// TIA Portal V20 export
FUNCTION "ManOperationCm_typeTwoWayActuatorInterface" : Void   // FC65, LAD
// stored: SetENOAutomatically false
   VAR_INPUT
      disableUnit : Bool;
   END_VAR
   VAR_OUTPUT
      Status : Word;
      errorID : Word;
   END_VAR
   VAR_IN_OUT
      manualOperationEm : "LAF_typeManEm";
      manualOperationEmArea : "LAF_typeManOperationArea";
      manualOperationCms : "LAF_typeManOperation";
      twoWayAcutor : "LBC_typeTwoWayActuatorInterface";
   END_VAR
BEGIN

REGION Network 1: Manual Operation Cm - typeTwoWayActuatorInterface
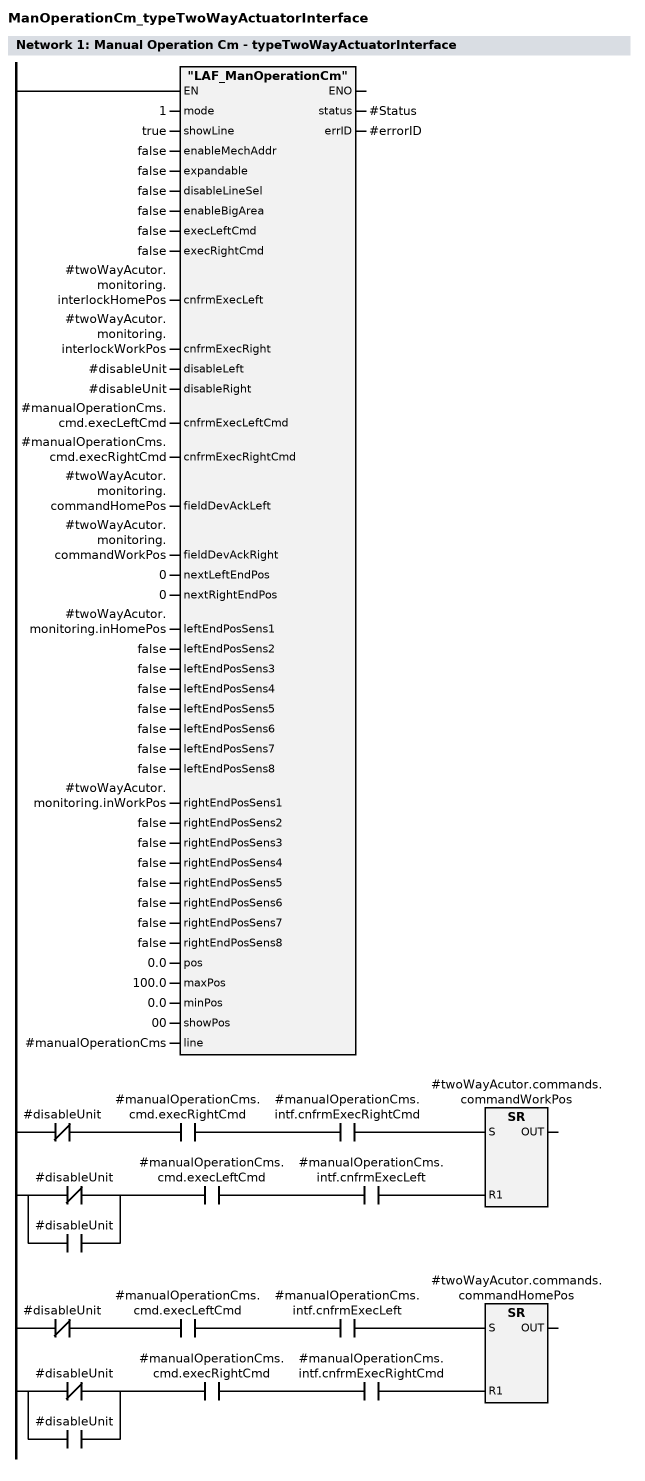
   RUNG wire#powerrail
      "LAF_ManOperationCm"(mode := 1, showLine := true, enableMechAddr := false, expandable := false, disableLineSel := false, enableBigArea := false, execLeftCmd := false, execRightCmd := false, cnfrmExecLeft := #twoWayAcutor.monitoring.interlockHomePos, cnfrmExecRight := #twoWayAcutor.monitoring.interlockWorkPos, disableLeft := #disableUnit, disableRight := #disableUnit, cnfrmExecLeftCmd := #manualOperationCms.cmd.execLeftCmd, cnfrmExecRightCmd := #manualOperationCms.cmd.execRightCmd, fieldDevAckLeft := #twoWayAcutor.monitoring.commandHomePos, fieldDevAckRight := #twoWayAcutor.monitoring.commandWorkPos, nextLeftEndPos := 0, nextRightEndPos := 0, leftEndPosSens1 := #twoWayAcutor.monitoring.inHomePos, leftEndPosSens2 := false, leftEndPosSens3 := false, leftEndPosSens4 := false, leftEndPosSens5 := false, leftEndPosSens6 := false, leftEndPosSens7 := false, leftEndPosSens8 := false, rightEndPosSens1 := #twoWayAcutor.monitoring.inWorkPos, rightEndPosSens2 := false, rightEndPosSens3 := false, rightEndPosSens4 := false, rightEndPosSens5 := false, rightEndPosSens6 := false, rightEndPosSens7 := false, rightEndPosSens8 := false, pos := 0.0, maxPos := 100.0, minPos := 0.0, showPos := 00, line := #manualOperationCms, status => #Status, errID => #errorID)
   END_RUNG
   RUNG wire#powerrail
      I_Contact( #disableUnit )
      Contact( #manualOperationCms.cmd.execRightCmd )
      Contact( #manualOperationCms.intf.cnfrmExecRightCmd )
      S_SR(operand := #twoWayAcutor.commands.commandWorkPos, r1 := wire#w2)
   END_RUNG
   RUNG wire#powerrail
      I_Contact( #disableUnit )
      wire#w1
      Contact( #manualOperationCms.cmd.execLeftCmd )
      Contact( #manualOperationCms.intf.cnfrmExecLeft )
   END_RUNG wire#w2
   RUNG wire#powerrail
      Contact( #disableUnit )
   END_RUNG wire#w1
   RUNG wire#powerrail
      I_Contact( #disableUnit )
      Contact( #manualOperationCms.cmd.execLeftCmd )
      Contact( #manualOperationCms.intf.cnfrmExecLeft )
      S_SR(operand := #twoWayAcutor.commands.commandHomePos, r1 := wire#w4)
   END_RUNG
   RUNG wire#powerrail
      I_Contact( #disableUnit )
      wire#w3
      Contact( #manualOperationCms.cmd.execRightCmd )
      Contact( #manualOperationCms.intf.cnfrmExecRightCmd )
   END_RUNG wire#w4
   RUNG wire#powerrail
      Contact( #disableUnit )
   END_RUNG wire#w3
   // the same network as SCL:
   "LAF_ManOperationCm"(mode := 1,
                        showLine := true,
                        enableMechAddr := false,
                        expandable := false,
                        disableLineSel := false,
                        enableBigArea := false,
                        execLeftCmd := false,
                        execRightCmd := false,
                        cnfrmExecLeft := #twoWayAcutor.monitoring.interlockHomePos,
                        cnfrmExecRight := #twoWayAcutor.monitoring.interlockWorkPos,
                        disableLeft := #disableUnit,
                        disableRight := #disableUnit,
                        cnfrmExecLeftCmd := #manualOperationCms.cmd.execLeftCmd,
                        cnfrmExecRightCmd := #manualOperationCms.cmd.execRightCmd,
                        fieldDevAckLeft := #twoWayAcutor.monitoring.commandHomePos,
                        fieldDevAckRight := #twoWayAcutor.monitoring.commandWorkPos,
                        nextLeftEndPos := 0,
                        nextRightEndPos := 0,
                        leftEndPosSens1 := #twoWayAcutor.monitoring.inHomePos,
                        leftEndPosSens2 := false,
                        leftEndPosSens3 := false,
                        leftEndPosSens4 := false,
                        leftEndPosSens5 := false,
                        leftEndPosSens6 := false,
                        leftEndPosSens7 := false,
                        leftEndPosSens8 := false,
                        rightEndPosSens1 := #twoWayAcutor.monitoring.inWorkPos,
                        rightEndPosSens2 := false,
                        rightEndPosSens3 := false,
                        rightEndPosSens4 := false,
                        rightEndPosSens5 := false,
                        rightEndPosSens6 := false,
                        rightEndPosSens7 := false,
                        rightEndPosSens8 := false,
                        pos := 0.0,
                        maxPos := 100.0,
                        minPos := 0.0,
                        showPos := 00,
                        line := #manualOperationCms,
                        status => #Status,
                        errID => #errorID);
   IF NOT #disableUnit AND #manualOperationCms.cmd.execRightCmd AND #manualOperationCms.intf.cnfrmExecRightCmd THEN
       #twoWayAcutor.commands.commandWorkPos := TRUE;   // SR flip-flop
   END_IF;
   IF (NOT #disableUnit OR #disableUnit) AND #manualOperationCms.cmd.execLeftCmd AND #manualOperationCms.intf.cnfrmExecLeft THEN
       #twoWayAcutor.commands.commandWorkPos := FALSE;
   END_IF;
   IF NOT #disableUnit AND #manualOperationCms.cmd.execLeftCmd AND #manualOperationCms.intf.cnfrmExecLeft THEN
       #twoWayAcutor.commands.commandHomePos := TRUE;   // SR flip-flop
   END_IF;
   IF (NOT #disableUnit OR #disableUnit) AND #manualOperationCms.cmd.execRightCmd AND #manualOperationCms.intf.cnfrmExecRightCmd THEN
       #twoWayAcutor.commands.commandHomePos := FALSE;
   END_IF;
END_REGION
END_FUNCTION
